// TIA Portal V19 export
VAR_GLOBAL   // PLC tag table "LB301"
   LB301_ScaricoSemilavorati_DX_Pb_Aux1 AT %I251.3 : Bool;   // 342SH1
   LB301_ScaricoSemilavorati_DX_Pb_Aux2 AT %I251.4 : Bool;   // 342SH2
   LB301_ScaricoSemilavorati_DX_Lp_Aux1 AT %Q250.7 : Bool;   // 342SH1
   LB301_ScaricoSemilavorati_DX_Lp_Aux2 AT %Q251.0 : Bool;   // 342SH2
END_VAR
